{attribute 'qualified_only'}
{attribute 'strict'}
{attribute 'to_string'}
TYPE PositingBarAlignmentDirection :
(
	AlingmentLeft := 0,
	AlingmentRight
);
END_TYPE

(* stored: Version 1.1.0.1
   DUT PositingBarAlignmentDirection: Id {3921d5cb-3fe0-41bf-95da-920f128ee3a3} *)
